// TIA Portal V18 export
DATA_BLOCK "AutoProcessDataPopUp_DB"   // DB2
VERSION : 0.1
// stored: AutoNumber true, DBAccessibleFromOPCUA true, DBAccessibleFromWebserver true, InstanceOfName AutoProcessDataPopUp, InstanceOfType FB
"AutoProcessDataPopUp"
   // VAR_IN_OUT
   //    idx { ExternalAccessible := 'False'; ExternalVisible := 'False'; ExternalWritable := 'False'} : Int;
   // END_VAR
BEGIN
END_DATA_BLOCK
